KUKA KRL program: PROJET_PROFILO.src, PROJET_PROFILO.dat

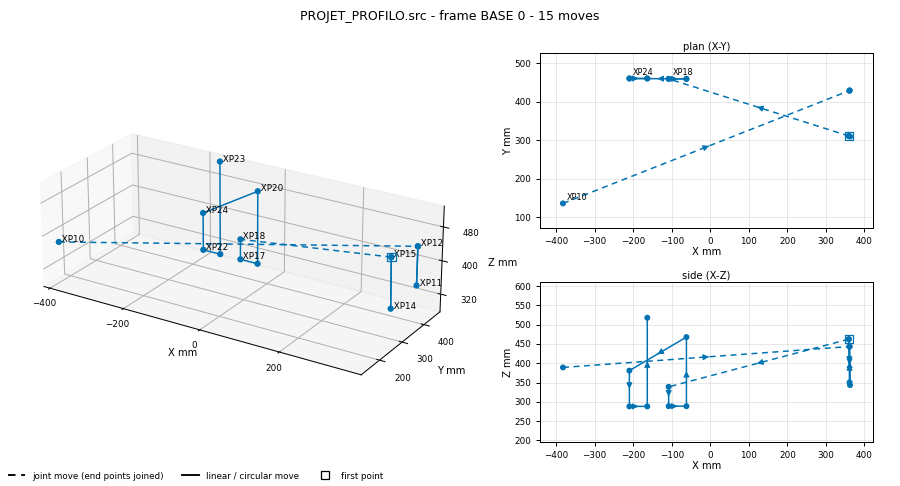
[picture p0: tool path of PROJET_PROFILO.src in frame BASE 0, 15 of 24 moves have a stored position in this frame; points joined in program order, loops and branches not executed]
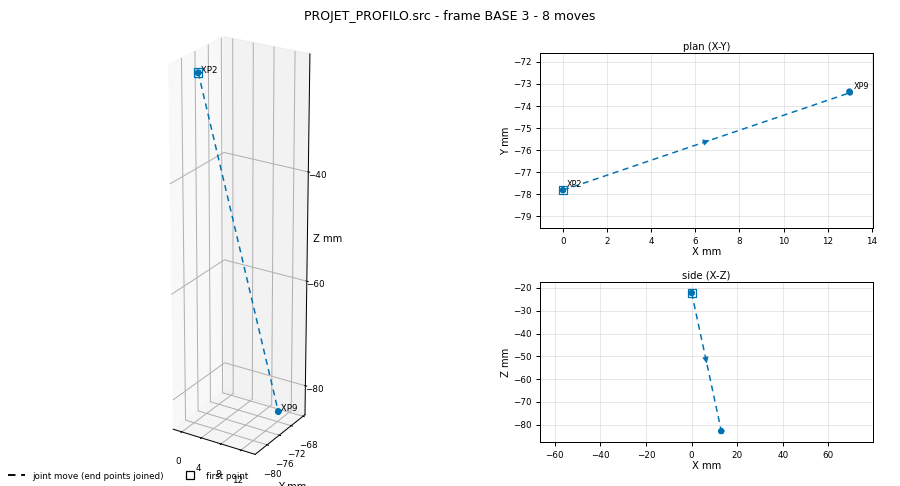
[picture p1: tool path of PROJET_PROFILO.src in frame BASE 3, 8 of 24 moves have a stored position in this frame; points joined in program order, loops and branches not executed]
--- PROJET_PROFILO.src ---
&ACCESS RVO
&REL 258
&PARAM TEMPLATE = C:\KRC\Roboter\Template\vorgabe
&PARAM EDITMASK = *
DEF PROJET_PROFILO( )
EXTFCT BOOL SEND(INT:OUT, STATE_T:OUT, STATE_T:OUT, MODUS_T:OUT)
EXTFCT BOOL RECEIVE(INT:OUT, STATE_T:OUT, STATE_T:OUT, MODUS_T:OUT, FRAME:OUT)
EXTFCT BOOL RECV_CHAR(INT:OUT, STATE_T:OUT, STATE_T:OUT, MODUS_T:OUT, CHAR:OUT)
EXTFCT BOOL RECV_DOUBLE(INT:OUT, STATE_T:OUT, STATE_T:OUT, MODUS_T:OUT, REAL:OUT)
EXTFCT BOOL SEND_CHAR(INT:OUT, STATE_T:OUT, STATE_T:OUT, MODUS_T:OUT, CHAR:IN)
EXTFCT BOOL PRENDRE_PROFILE(INT:OUT, STATE_T:OUT, STATE_T:OUT, MODUS_T:OUT, CHAR:OUT)

DECL INT HANDLE
DECL STATE_T SR_T
DECL STATE_T SC_T
DECL MODUS_T MR_T
DECL CHAR IN_CHAR
DECL CHAR OUT_CHAR
DECL BOOL R1

;FOLD INI
  ;FOLD BASISTECH INI
    GLOBAL INTERRUPT DECL 3 WHEN $STOPMESS==TRUE DO IR_STOPM ( )
    INTERRUPT ON 3
    BAS (#INITMOV,0 )
  ;ENDFOLD (BASISTECH INI)
  ;FOLD USER INI
    ;Make your modifications here

  ;ENDFOLD (USER INI)
;ENDFOLD (INI)
; initialization
IN_CHAR = " "
OUT_CHAR = " "
MR_T = #ABS

;FOLD PTP HOME  Vel= 10 % PDAT24;%{PE}%R 5.4.37,%MKUKATPBASIS,%CMOVE,%VPTP,%P 1:PTP, 2:HOME, 3:, 5:10, 7:PDAT24
$BWDSTART=FALSE
PDAT_ACT=PPDAT24
FDAT_ACT=FHOME
BAS(#PTP_PARAMS,10)
$H_POS=XHOME
PTP XHOME
;ENDFOLD

LOOP
;FOLD PULSE 27 'lacher'  State= TRUE   Time= 0.5 sec;%{PE}%R 5.4.37,%MKUKATPBASIS,%COUT,%VPULSE,%P 2:27, 3:lacher, 5:TRUE, 6:, 8:0.5
PULSE($OUT[27], TRUE,0.5)
;ENDFOLD
;FOLD WAIT Time= 1 sec;%{PE}%R 5.4.37,%MKUKATPBASIS,%CWAIT,%VWAIT,%P 2:1
WAIT SEC 1
;ENDFOLD
;FOLD PULSE 25 'prendre'  State= TRUE   Time= 0.5 sec;%{PE}%R 5.4.37,%MKUKATPBASIS,%COUT,%VPULSE,%P 2:25, 3:prendre, 5:TRUE, 6:, 8:0.5
PULSE($OUT[25], TRUE,0.5)
;ENDFOLD

; wait GO signal from PC
WHILE (IN_CHAR <> 71)
   R1 = RECV_CHAR(HANDLE, SR_T, SC_T, MR_T, IN_CHAR)
ENDWHILE

; go grab the cube
;FOLD PTP P15  Vel= 20 % PDAT28 Tool[3]:pince Base[0];%{PE}%R 5.4.37,%MKUKATPBASIS,%CMOVE,%VPTP,%P 1:PTP, 2:P15, 3:, 5:20, 7:PDAT28
$BWDSTART=FALSE
PDAT_ACT=PPDAT28
FDAT_ACT=FP15
BAS(#PTP_PARAMS,20)
PTP XP15
;ENDFOLD
;FOLD LIN P14  Vel= 0.1 m/s CPDAT18 Tool[3]:pince Base[0];%{PE}%R 5.4.37,%MKUKATPBASIS,%CMOVE,%VLIN,%P 1:LIN, 2:P14, 3:, 5:0.1, 7:CPDAT18
$BWDSTART=FALSE
LDAT_ACT=LCPDAT18
FDAT_ACT=FP14
BAS(#CP_PARAMS,0.1)
LIN XP14
;ENDFOLD
;FOLD PULSE 27 'lacher'  State= TRUE   Time= 0.5 sec;%{PE}%R 5.4.37,%MKUKATPBASIS,%COUT,%VPULSE,%P 2:27, 3:lacher, 5:TRUE, 6:, 8:0.5
PULSE($OUT[27], TRUE,0.5)
;ENDFOLD
;FOLD LIN P16  Vel= 0.2 m/s CPDAT19 Tool[3]:pince Base[0];%{PE}%R 5.4.37,%MKUKATPBASIS,%CMOVE,%VLIN,%P 1:LIN, 2:P16, 3:, 5:0.2, 7:CPDAT19
$BWDSTART=FALSE
LDAT_ACT=LCPDAT19
FDAT_ACT=FP16
BAS(#CP_PARAMS,0.2)
LIN XP16
;ENDFOLD

; cube taken, now go flip the cube
;FOLD PTP P18  Vel= 20 % PDAT29 Tool[3]:pince Base[0];%{PE}%R 5.4.37,%MKUKATPBASIS,%CMOVE,%VPTP,%P 1:PTP, 2:P18, 3:, 5:20, 7:PDAT29
$BWDSTART=FALSE
PDAT_ACT=PPDAT29
FDAT_ACT=FP18
BAS(#PTP_PARAMS,20)
PTP XP18
;ENDFOLD
;FOLD LIN P17  Vel= 0.1 m/s CPDAT20 Tool[3]:pince Base[0];%{PE}%R 5.4.37,%MKUKATPBASIS,%CMOVE,%VLIN,%P 1:LIN, 2:P17, 3:, 5:0.1, 7:CPDAT20
$BWDSTART=FALSE
LDAT_ACT=LCPDAT20
FDAT_ACT=FP17
BAS(#CP_PARAMS,0.1)
LIN XP17
;ENDFOLD
;FOLD PULSE 25 'prendre'  State= TRUE   Time= 0.5 sec;%{PE}%R 5.4.37,%MKUKATPBASIS,%COUT,%VPULSE,%P 2:25, 3:prendre, 5:TRUE, 6:, 8:0.5
PULSE($OUT[25], TRUE,0.5)
;ENDFOLD
;FOLD LIN P19  Vel= 0.1 m/s CPDAT21 Tool[3]:pince Base[0];%{PE}%R 5.4.37,%MKUKATPBASIS,%CMOVE,%VLIN,%P 1:LIN, 2:P19, 3:, 5:0.1, 7:CPDAT21
$BWDSTART=FALSE
LDAT_ACT=LCPDAT21
FDAT_ACT=FP19
BAS(#CP_PARAMS,0.1)
LIN XP19
;ENDFOLD
;FOLD LIN P20 CONT Vel= 0.1 m/s CPDAT24 Tool[3]:pince Base[0];%{PE}%R 5.4.37,%MKUKATPBASIS,%CMOVE,%VLIN,%P 1:LIN, 2:P20, 3:C_DIS, 5:0.1, 7:CPDAT24
$BWDSTART=FALSE
LDAT_ACT=LCPDAT24
FDAT_ACT=FP20
BAS(#CP_PARAMS,0.1)
LIN XP20 C_DIS
;ENDFOLD
;FOLD PULSE 27 'lacher'  State= TRUE   Time= 0.5 sec;%{PE}%R 5.4.37,%MKUKATPBASIS,%COUT,%VPULSE,%P 2:27, 3:lacher, 5:TRUE, 6:, 8:0.5
PULSE($OUT[27], TRUE,0.5)
;ENDFOLD
;FOLD LIN P24 CONT Vel= 0.1 m/s CPDAT26 Tool[3]:pince Base[0];%{PE}%R 5.4.37,%MKUKATPBASIS,%CMOVE,%VLIN,%P 1:LIN, 2:P24, 3:C_DIS, 5:0.1, 7:CPDAT26
$BWDSTART=FALSE
LDAT_ACT=LCPDAT26
FDAT_ACT=FP24
BAS(#CP_PARAMS,0.1)
LIN XP24 C_DIS
;ENDFOLD
;FOLD LIN P22  Vel= 0.1 m/s CPDAT25 Tool[3]:pince Base[0];%{PE}%R 5.4.37,%MKUKATPBASIS,%CMOVE,%VLIN,%P 1:LIN, 2:P22, 3:, 5:0.1, 7:CPDAT25
$BWDSTART=FALSE
LDAT_ACT=LCPDAT25
FDAT_ACT=FP22
BAS(#CP_PARAMS,0.1)
LIN XP22
;ENDFOLD
;FOLD LIN P21  Vel= 0.1 m/s CPDAT22 Tool[3]:pince Base[0];%{PE}%R 5.4.37,%MKUKATPBASIS,%CMOVE,%VLIN,%P 1:LIN, 2:P21, 3:, 5:0.1, 7:CPDAT22
$BWDSTART=FALSE
LDAT_ACT=LCPDAT22
FDAT_ACT=FP21
BAS(#CP_PARAMS,0.1)
LIN XP21
;ENDFOLD
;FOLD PULSE 25 'prendre'  State= TRUE   Time= 0.5 sec;%{PE}%R 5.4.37,%MKUKATPBASIS,%COUT,%VPULSE,%P 2:25, 3:prendre, 5:TRUE, 6:, 8:0.5
PULSE($OUT[25], TRUE,0.5)
;ENDFOLD
;FOLD LIN P23 CONT Vel= 0.1 m/s CPDAT23 Tool[3]:pince Base[0];%{PE}%R 5.4.37,%MKUKATPBASIS,%CMOVE,%VLIN,%P 1:LIN, 2:P23, 3:C_DIS, 5:0.1, 7:CPDAT23
$BWDSTART=FALSE
LDAT_ACT=LCPDAT23
FDAT_ACT=FP23
BAS(#CP_PARAMS,0.1)
LIN XP23 C_DIS
;ENDFOLD

; wait GO signal from PC
WHILE (IN_CHAR <> 71)
   R1 = RECV_CHAR(HANDLE, SR_T, SC_T, MR_T, IN_CHAR)
ENDWHILE

; go to points and take profiles
;FOLD PTP P2  Vel= 20 % PDAT19 Tool[3]:pince Base[3]:profilometre;%{PE}%R 5.4.37,%MKUKATPBASIS,%CMOVE,%VPTP,%P 1:PTP, 2:P2, 3:, 5:20, 7:PDAT19
$BWDSTART=FALSE
PDAT_ACT=PPDAT19
FDAT_ACT=FP2
BAS(#PTP_PARAMS,20)
PTP XP2
;ENDFOLD
R1 = PRENDRE_PROFILE(HANDLE, SR_T, SC_T, MR_T, IN_CHAR)
;FOLD PTP P6  Vel= 20 % PDAT20 Tool[3]:pince Base[3]:profilometre;%{PE}%R 5.4.37,%MKUKATPBASIS,%CMOVE,%VPTP,%P 1:PTP, 2:P6, 3:, 5:20, 7:PDAT20
$BWDSTART=FALSE
PDAT_ACT=PPDAT20
FDAT_ACT=FP6
BAS(#PTP_PARAMS,20)
PTP XP6
;ENDFOLD
R1 = PRENDRE_PROFILE(HANDLE, SR_T, SC_T, MR_T, IN_CHAR)
;FOLD PTP P7  Vel= 20 % PDAT21 Tool[3]:pince Base[3]:profilometre;%{PE}%R 5.4.37,%MKUKATPBASIS,%CMOVE,%VPTP,%P 1:PTP, 2:P7, 3:, 5:20, 7:PDAT21
$BWDSTART=FALSE
PDAT_ACT=PPDAT21
FDAT_ACT=FP7
BAS(#PTP_PARAMS,20)
PTP XP7
;ENDFOLD
R1 = PRENDRE_PROFILE(HANDLE, SR_T, SC_T, MR_T, IN_CHAR)
;FOLD PTP P8  Vel= 20 % PDAT22 Tool[3]:pince Base[3]:profilometre;%{PE}%R 5.4.37,%MKUKATPBASIS,%CMOVE,%VPTP,%P 1:PTP, 2:P8, 3:, 5:20, 7:PDAT22
$BWDSTART=FALSE
PDAT_ACT=PPDAT22
FDAT_ACT=FP8
BAS(#PTP_PARAMS,20)
PTP XP8
;ENDFOLD
R1 = PRENDRE_PROFILE(HANDLE, SR_T, SC_T, MR_T, IN_CHAR)

; upper face, scanned 4 times with different angles
;FOLD PTP P9  Vel= 20 % PDAT23 Tool[3]:pince Base[3]:profilometre;%{PE}%R 5.4.37,%MKUKATPBASIS,%CMOVE,%VPTP,%P 1:PTP, 2:P9, 3:, 5:20, 7:PDAT23
$BWDSTART=FALSE
PDAT_ACT=PPDAT23
FDAT_ACT=FP9
BAS(#PTP_PARAMS,20)
PTP XP9
;ENDFOLD
R1 = PRENDRE_PROFILE(HANDLE, SR_T, SC_T, MR_T, IN_CHAR)
;FOLD PTP P26  Vel= 20 % PDAT34 Tool[3]:pince Base[3]:profilometre;%{PE}%R 5.4.37,%MKUKATPBASIS,%CMOVE,%VPTP,%P 1:PTP, 2:P26, 3:, 5:20, 7:PDAT34
$BWDSTART=FALSE
PDAT_ACT=PPDAT34
FDAT_ACT=FP26
BAS(#PTP_PARAMS,20)
PTP XP26
;ENDFOLD
R1 = PRENDRE_PROFILE(HANDLE, SR_T, SC_T, MR_T, IN_CHAR)
;FOLD PTP P25  Vel= 20 % PDAT33 Tool[3]:pince Base[3]:profilometre;%{PE}%R 5.4.37,%MKUKATPBASIS,%CMOVE,%VPTP,%P 1:PTP, 2:P25, 3:, 5:20, 7:PDAT33
$BWDSTART=FALSE
PDAT_ACT=PPDAT33
FDAT_ACT=FP25
BAS(#PTP_PARAMS,20)
PTP XP25
;ENDFOLD
R1 = PRENDRE_PROFILE(HANDLE, SR_T, SC_T, MR_T, IN_CHAR)
;FOLD PTP P27  Vel= 20 % PDAT35 Tool[3]:pince Base[3]:profilometre;%{PE}%R 5.4.37,%MKUKATPBASIS,%CMOVE,%VPTP,%P 1:PTP, 2:P27, 3:, 5:20, 7:PDAT35
$BWDSTART=FALSE
PDAT_ACT=PPDAT35
FDAT_ACT=FP27
BAS(#PTP_PARAMS,20)
PTP XP27
;ENDFOLD
R1 = PRENDRE_PROFILE(HANDLE, SR_T, SC_T, MR_T, IN_CHAR)

; send EXIT to PC
R1 = SEND_CHAR(HANDLE, SR_T, SC_T, MR_T, 88)

; wait for PC tells part conform or not
WHILE (IN_CHAR <> 78) AND (IN_CHAR <> 89)
   R1 = RECV_CHAR(HANDLE, SR_T, SC_T, MR_T, IN_CHAR)
ENDWHILE

; part not conform
IF IN_CHAR == 78 THEN
;FOLD PTP P10  Vel= 20 % PDAT25 Tool[3]:pince Base[0];%{PE}%R 5.4.37,%MKUKATPBASIS,%CMOVE,%VPTP,%P 1:PTP, 2:P10, 3:, 5:20, 7:PDAT25
$BWDSTART=FALSE
PDAT_ACT=PPDAT25
FDAT_ACT=FP10
BAS(#PTP_PARAMS,20)
PTP XP10
;ENDFOLD
;FOLD PULSE 27 'lacher'  State= TRUE   Time= 0.5 sec;%{PE}%R 5.4.37,%MKUKATPBASIS,%COUT,%VPULSE,%P 2:27, 3:lacher, 5:TRUE, 6:, 8:0.5
PULSE($OUT[27], TRUE,0.5)
;ENDFOLD
ENDIF

; part conform
IF IN_CHAR == 89 THEN
;FOLD PTP P12  Vel= 20 % PDAT26 Tool[3]:pince Base[0];%{PE}%R 5.4.37,%MKUKATPBASIS,%CMOVE,%VPTP,%P 1:PTP, 2:P12, 3:, 5:20, 7:PDAT26
$BWDSTART=FALSE
PDAT_ACT=PPDAT26
FDAT_ACT=FP12
BAS(#PTP_PARAMS,20)
PTP XP12
;ENDFOLD
;FOLD LIN P11  Vel= 0.1 m/s CPDAT17 Tool[3]:pince Base[0];%{PE}%R 5.4.37,%MKUKATPBASIS,%CMOVE,%VLIN,%P 1:LIN, 2:P11, 3:, 5:0.1, 7:CPDAT17
$BWDSTART=FALSE
LDAT_ACT=LCPDAT17
FDAT_ACT=FP11
BAS(#CP_PARAMS,0.1)
LIN XP11
;ENDFOLD
;FOLD PULSE 27 'lacher'  State= TRUE   Time= 0.5 sec;%{PE}%R 5.4.37,%MKUKATPBASIS,%COUT,%VPULSE,%P 2:27, 3:lacher, 5:TRUE, 6:, 8:0.5
PULSE($OUT[27], TRUE,0.5)
;ENDFOLD
;FOLD LIN P13  Vel= 0.2 m/s CPDAT27 Tool[3]:pince Base[0];%{PE}%R 5.4.37,%MKUKATPBASIS,%CMOVE,%VLIN,%P 1:LIN, 2:P13, 3:, 5:0.2, 7:CPDAT27
$BWDSTART=FALSE
LDAT_ACT=LCPDAT27
FDAT_ACT=FP13
BAS(#CP_PARAMS,0.2)
LIN XP13
;ENDFOLD
ENDIF

ENDLOOP
END

--- PROJET_PROFILO.dat ---
&ACCESS RVO
&REL 258
&PARAM TEMPLATE = C:\KRC\Roboter\Template\vorgabe
&PARAM EDITMASK = *
DEFDAT  PROJET_PROFILO
;FOLD EXTERNAL DECLARATIONS;%{PE}%MKUKATPBASIS,%CEXT,%VCOMMON,%P
;FOLD BASISTECH EXT;%{PE}%MKUKATPBASIS,%CEXT,%VEXT,%P
EXT  BAS (BAS_COMMAND  :IN,REAL  :IN )
DECL INT SUCCESS
;ENDFOLD (BASISTECH EXT)
;FOLD USER EXT;%{E}%MKUKATPUSER,%CEXT,%VEXT,%P
;Make here your modifications

;ENDFOLD (USER EXT)
;ENDFOLD (EXTERNAL DECLERATIONS)
DECL BASIS_SUGG_T LAST_BASIS={POINT1[] "P27                     ",POINT2[] "P27                     ",CP_PARAMS[] "CPDAT26                 ",PTP_PARAMS[] "PDAT35                  ",CONT[] "                        ",CP_VEL[] "0.005                   ",PTP_VEL[] "20                      ",SPL_NAME[] "S0                      "}
DECL E6POS XP1={X 3.04208207,Y 411.683594,Z 361.17569,A 167.849899,B 89.528801,C 152.8974,S 2,T 43,E1 0.0,E2 0.0,E3 0.0,E4 0.0,E5 0.0,E6 0.0}
DECL FDAT FP1={TOOL_NO 2,BASE_NO 0,IPO_FRAME #BASE,POINT2[] " "}
DECL PDAT PPDAT1={VEL 100.0,ACC 100.0,APO_DIST 100.0}
DECL PDAT PPDAT2={VEL 100.0,ACC 100.0,APO_DIST 100.0}
DECL PDAT PPDAT3={VEL 100.0,ACC 100.0,APO_DIST 100.0}
DECL PDAT PPDAT4={VEL 100.0,ACC 100.0,APO_DIST 100.0}
DECL PDAT PPDAT5={VEL 100.0,ACC 100.0,APO_DIST 100.0}
DECL PDAT PPDAT6={VEL 100.0,ACC 100.0,APO_DIST 100.0}
DECL PDAT PPDAT7={VEL 100.0,ACC 100.0,APO_DIST 100.0}
DECL E6POS XP99={X -85.5281525,Y 414.985596,Z 387.865997,A 88.0866013,B 87.5991135,C 97.2242432,S 2,T 35,E1 0.0,E2 0.0,E3 0.0,E4 0.0,E5 0.0,E6 0.0}
DECL FDAT FP99={TOOL_NO 2,BASE_NO 0,IPO_FRAME #BASE,POINT2[] " "}
DECL PDAT PPDAT8={VEL 100.0,ACC 100.0,APO_DIST 100.0}
DECL INT LAST_XP_POINT=9
DECL E6POS XNEW_POINT={X -251.468094,Y 292.194702,Z 631.135681,A 91.6703262,B -87.1333008,C -129.946304,S 2,T 43,E1 0.0,E2 0.0,E3 0.0,E4 0.0,E5 0.0,E6 0.0}
DECL FDAT FNEW_POINT={TOOL_NO 0,BASE_NO 0,IPO_FRAME #BASE,POINT2[] " "}
DECL LDAT LCPDAT1={VEL 2.0,ACC 100.0,APO_DIST 100.0,APO_FAC 50.0,ORI_TYP #VAR}
DECL LDAT LCPDAT2={VEL 2.0,ACC 100.0,APO_DIST 100.0,APO_FAC 50.0,ORI_TYP #VAR}
DECL E6POS XINITIAL_POS={X 352.895111,Y 300.94281,Z 673.360901,A -90.7709427,B -1.56862795,C -179.936905,S 2,T 35,E1 0.0,E2 0.0,E3 0.0,E4 0.0,E5 0.0,E6 0.0}
DECL FDAT FINITIAL_POS={TOOL_NO 0,BASE_NO 0,IPO_FRAME #BASE,POINT2[] " "}
DECL PDAT PPDAT9={VEL 100.0,ACC 100.0,APO_DIST 100.0}
DECL PDAT PPDAT10={VEL 100.0,ACC 100.0,APO_DIST 100.0}
DECL LDAT LCPDAT3={VEL 2.0,ACC 100.0,APO_DIST 100.0,APO_FAC 50.0,ORI_TYP #VAR}
DECL LDAT LCPDAT4={VEL 2.0,ACC 100.0,APO_DIST 100.0,APO_FAC 50.0,ORI_TYP #VAR}
DECL LDAT LCPDAT5={VEL 2.0,ACC 100.0,APO_DIST 100.0,APO_FAC 50.0,ORI_TYP #VAR}
DECL LDAT LCPDAT6={VEL 2.0,ACC 100.0,APO_DIST 100.0,APO_FAC 50.0,ORI_TYP #VAR}
DECL LDAT LCPDAT7={VEL 2.0,ACC 100.0,APO_DIST 100.0,APO_FAC 50.0,ORI_TYP #VAR}
DECL E6POS XNEW_POINT_LIN_FAST={X -60.5829201,Y 419.159485,Z 498.605988,A 67.120079,B -2.27553606,C -179.295593,S 2,T 35,E1 0.0,E2 0.0,E3 0.0,E4 0.0,E5 0.0,E6 0.0}
DECL FDAT FNEW_POINT_LIN_FAST={TOOL_NO 0,BASE_NO 0,IPO_FRAME #BASE,POINT2[] " "}
DECL E6POS XNEW_POINT_LIN_SLOW={X -60.5829201,Y 419.159485,Z 498.605988,A 67.120079,B -2.27553606,C -179.295593,S 2,T 35,E1 0.0,E2 0.0,E3 0.0,E4 0.0,E5 0.0,E6 0.0}
DECL FDAT FNEW_POINT_LIN_SLOW={TOOL_NO 0,BASE_NO 0,IPO_FRAME #BASE,POINT2[] " "}
DECL PDAT PPDAT11={VEL 100.0,ACC 100.0,APO_DIST 100.0}
DECL PDAT PPDAT12={VEL 100.0,ACC 100.0,APO_DIST 100.0}
DECL LDAT LCPDAT8={VEL 2.0,ACC 100.0,APO_DIST 100.0,APO_FAC 50.0,ORI_TYP #VAR}
DECL LDAT LCPDAT9={VEL 2.0,ACC 100.0,APO_DIST 100.0,APO_FAC 50.0,ORI_TYP #VAR}
DECL PDAT PPDAT13={VEL 100.0,ACC 100.0,APO_DIST 100.0}
DECL E6POS XP2={X 0.00264483108,Y -77.8235779,Z -22.1945,A -153.933197,B -88.8520432,C 65.1572266,S 6,T 59,E1 0.0,E2 0.0,E3 0.0,E4 0.0,E5 0.0,E6 0.0}
DECL FDAT FP2={TOOL_NO 3,BASE_NO 3,IPO_FRAME #BASE,POINT2[] " "}
DECL PDAT PPDAT14={VEL 100.0,ACC 100.0,APO_DIST 100.0}
DECL E6POS XP3={X 0.211270601,Y 480.734589,Z 566.639587,A -94.440567,B 2.11090398,C 90.3766479,S 6,T 51,E1 0.0,E2 0.0,E3 0.0,E4 0.0,E5 0.0,E6 0.0}
DECL FDAT FP3={TOOL_NO 0,BASE_NO 0,IPO_FRAME #BASE,POINT2[] " "}
DECL LDAT LCPDAT10={VEL 2.0,ACC 100.0,APO_DIST 100.0,APO_FAC 50.0,ORI_TYP #VAR}
DECL E6POS XP4={X 0.211270601,Y 480.734589,Z 566.639587,A -94.440567,B 2.11090398,C 90.3766479,S 6,T 51,E1 0.0,E2 0.0,E3 0.0,E4 0.0,E5 0.0,E6 0.0}
DECL FDAT FP4={TOOL_NO 0,BASE_NO 0,IPO_FRAME #BASE,POINT2[] " "}
DECL LDAT LCPDAT11={VEL 2.0,ACC 100.0,APO_DIST 100.0,APO_FAC 50.0,ORI_TYP #VAR}
DECL E6POS XP5={X 47.832859,Y 50.5500603,Z -203.236404,A -94.440567,B 2.11090398,C 90.3766479,S 6,T 51,E1 0.0,E2 0.0,E3 0.0,E4 0.0,E5 0.0,E6 0.0}
DECL FDAT FP5={TOOL_NO 3,BASE_NO 3,IPO_FRAME #BASE,POINT2[] " "}
DECL LDAT LCPDAT12={VEL 2.0,ACC 100.0,APO_DIST 100.0,APO_FAC 50.0,ORI_TYP #VAR}
DECL E6POS XP6={X 0.00117324002,Y -77.8127594,Z -22.2087898,A -179.498199,B -0.486956209,C 91.2150726,S 6,T 27,E1 0.0,E2 0.0,E3 0.0,E4 0.0,E5 0.0,E6 0.0}
DECL FDAT FP6={TOOL_NO 3,BASE_NO 3,IPO_FRAME #BASE,POINT2[] " "}
DECL PDAT PPDAT15={VEL 100.0,ACC 100.0,APO_DIST 100.0}
DECL E6POS XP7={X 0.00117345597,Y -77.8127594,Z -22.2087898,A -19.7653904,B 88.5158768,C -108.539902,S 6,T 27,E1 0.0,E2 0.0,E3 0.0,E4 0.0,E5 0.0,E6 0.0}
DECL FDAT FP7={TOOL_NO 3,BASE_NO 3,IPO_FRAME #BASE,POINT2[] " "}
DECL PDAT PPDAT16={VEL 100.0,ACC 100.0,APO_DIST 100.0}
DECL E6POS XP8={X 0.00117460405,Y -77.8127594,Z -22.2087898,A -0.501615882,B 0.0515326709,C -88.7053375,S 6,T 59,E1 0.0,E2 0.0,E3 0.0,E4 0.0,E5 0.0,E6 0.0}
DECL FDAT FP8={TOOL_NO 3,BASE_NO 3,IPO_FRAME #BASE,POINT2[] " "}
DECL PDAT PPDAT17={VEL 100.0,ACC 100.0,APO_DIST 100.0}
DECL LDAT LCPDAT13={VEL 2.0,ACC 100.0,APO_DIST 100.0,APO_FAC 50.0,ORI_TYP #VAR}
DECL LDAT LCPDAT14={VEL 2.0,ACC 100.0,APO_DIST 100.0,APO_FAC 50.0,ORI_TYP #VAR}
DECL LDAT LCPDAT15={VEL 2.0,ACC 100.0,APO_DIST 100.0,APO_FAC 50.0,ORI_TYP #VAR}
DECL LDAT LCPDAT16={VEL 2.0,ACC 100.0,APO_DIST 100.0,APO_FAC 50.0,ORI_TYP #VAR}
DECL PDAT PPDAT18={VEL 100.0,ACC 100.0,APO_DIST 100.0}
DECL PDAT PPDAT19={VEL 100.0,ACC 100.0,APO_DIST 100.0}
DECL PDAT PPDAT20={VEL 100.0,ACC 100.0,APO_DIST 100.0}
DECL PDAT PPDAT21={VEL 100.0,ACC 100.0,APO_DIST 100.0}
DECL PDAT PPDAT22={VEL 100.0,ACC 100.0,APO_DIST 100.0}
DECL E6POS XP9={X 13.0152302,Y -73.394043,Z -82.7755432,A -175.600098,B 1.09652495,C 26.9111309,S 6,T 59,E1 0.0,E2 0.0,E3 0.0,E4 0.0,E5 0.0,E6 0.0}
DECL FDAT FP9={TOOL_NO 3,BASE_NO 3,IPO_FRAME #BASE,POINT2[] " "}
DECL PDAT PPDAT23={VEL 100.0,ACC 100.0,APO_DIST 100.0}
DECL PDAT PPDAT24={VEL 100.0,ACC 100.0,APO_DIST 100.0}
DECL E6POS XP10={X -382.229797,Y 136.348206,Z 389.157715,A 87.4006577,B -1.75323403,C -177.311707,S 6,T 59,E1 0.0,E2 0.0,E3 0.0,E4 0.0,E5 0.0,E6 0.0}
DECL FDAT FP10={TOOL_NO 3,BASE_NO 0,IPO_FRAME #BASE,POINT2[] " "}
DECL PDAT PPDAT25={VEL 100.0,ACC 100.0,APO_DIST 100.0}
DECL E6POS XP11={X 361.469086,Y 429.168213,Z 350.290985,A 89.2297974,B -0.773940682,C -179.077301,S 2,T 43,E1 0.0,E2 0.0,E3 0.0,E4 0.0,E5 0.0,E6 0.0}
DECL FDAT FP11={TOOL_NO 3,BASE_NO 0,IPO_FRAME #BASE,POINT2[] " "}
DECL LDAT LCPDAT17={VEL 2.0,ACC 100.0,APO_DIST 100.0,APO_FAC 50.0,ORI_TYP #VAR}
DECL E6POS XP12={X 361.442413,Y 429.135406,Z 443.394714,A 89.2239227,B -0.758097708,C -179.062393,S 2,T 43,E1 0.0,E2 0.0,E3 0.0,E4 0.0,E5 0.0,E6 0.0}
DECL FDAT FP12={TOOL_NO 3,BASE_NO 0,IPO_FRAME #BASE,POINT2[] " "}
DECL PDAT PPDAT26={VEL 100.0,ACC 100.0,APO_DIST 100.0}
DECL E6POS XP13={X 361.442413,Y 429.135406,Z 443.394714,A 89.2239227,B -0.758097708,C -179.062393,S 2,T 43,E1 0.0,E2 0.0,E3 0.0,E4 0.0,E5 0.0,E6 0.0}
DECL FDAT FP13={TOOL_NO 3,BASE_NO 0,IPO_FRAME #BASE,POINT2[] " "}
DECL PDAT PPDAT27={VEL 100.0,ACC 100.0,APO_DIST 100.0}
DECL E6POS XP14={X 362.679688,Y 309.753906,Z 343.361603,A 179.220901,B -0.79322809,C 179.790802,S 2,T 43,E1 0.0,E2 0.0,E3 0.0,E4 0.0,E5 0.0,E6 0.0}
DECL FDAT FP14={TOOL_NO 3,BASE_NO 0,IPO_FRAME #BASE,POINT2[] " "}
DECL LDAT LCPDAT18={VEL 2.0,ACC 100.0,APO_DIST 100.0,APO_FAC 50.0,ORI_TYP #VAR}
DECL E6POS XP15={X 359.65799,Y 311.270905,Z 462.464996,A 179.216599,B -0.798424482,C 179.8069,S 2,T 43,E1 0.0,E2 0.0,E3 0.0,E4 0.0,E5 0.0,E6 0.0}
DECL FDAT FP15={TOOL_NO 3,BASE_NO 0,IPO_FRAME #BASE,POINT2[] " "}
DECL PDAT PPDAT28={VEL 100.0,ACC 100.0,APO_DIST 100.0}
DECL E6POS XP16={X 359.65799,Y 311.270905,Z 462.464996,A 179.216599,B -0.798424482,C 179.8069,S 2,T 43,E1 0.0,E2 0.0,E3 0.0,E4 0.0,E5 0.0,E6 0.0}
DECL FDAT FP16={TOOL_NO 3,BASE_NO 0,IPO_FRAME #BASE,POINT2[] " "}
DECL LDAT LCPDAT19={VEL 2.0,ACC 100.0,APO_DIST 100.0,APO_FAC 50.0,ORI_TYP #VAR}
DECL E6POS XP17={X -107.957001,Y 459.539398,Z 288.618195,A -89.8100433,B -0.0262975805,C 91.8582687,S 2,T 11,E1 0.0,E2 0.0,E3 0.0,E4 0.0,E5 0.0,E6 0.0}
DECL FDAT FP17={TOOL_NO 3,BASE_NO 0,IPO_FRAME #BASE,POINT2[] " "}
DECL LDAT LCPDAT20={VEL 2.0,ACC 100.0,APO_DIST 100.0,APO_FAC 50.0,ORI_TYP #VAR}
DECL E6POS XP18={X -107.951401,Y 459.55069,Z 338.765594,A -89.8116684,B -0.0291104,C 91.8583374,S 2,T 11,E1 0.0,E2 0.0,E3 0.0,E4 0.0,E5 0.0,E6 0.0}
DECL FDAT FP18={TOOL_NO 3,BASE_NO 0,IPO_FRAME #BASE,POINT2[] " "}
DECL PDAT PPDAT29={VEL 100.0,ACC 100.0,APO_DIST 100.0}
DECL E6POS XP19={X -61.8498192,Y 459.524506,Z 288.55069,A -89.8078079,B -0.0331712812,C 91.8604126,S 2,T 11,E1 0.0,E2 0.0,E3 0.0,E4 0.0,E5 0.0,E6 0.0}
DECL FDAT FP19={TOOL_NO 3,BASE_NO 0,IPO_FRAME #BASE,POINT2[] " "}
DECL LDAT LCPDAT21={VEL 2.0,ACC 100.0,APO_DIST 100.0,APO_FAC 50.0,ORI_TYP #VAR}
DECL E6POS XP20={X -61.852829,Y 459.462006,Z 467.888,A -89.7964706,B -0.0613530986,C 91.8438721,S 2,T 11,E1 0.0,E2 0.0,E3 0.0,E4 0.0,E5 0.0,E6 0.0}
DECL FDAT FP20={TOOL_NO 3,BASE_NO 0,IPO_FRAME #BASE,POINT2[] " "}
DECL PDAT PPDAT30={VEL 100.0,ACC 100.0,APO_DIST 100.0}
DECL E6POS XP21={X -163.422806,Y 460.499115,Z 288.062714,A -90.2210999,B -0.260996312,C -90.0108871,S 2,T 35,E1 0.0,E2 0.0,E3 0.0,E4 0.0,E5 0.0,E6 0.0}
DECL FDAT FP21={TOOL_NO 3,BASE_NO 0,IPO_FRAME #BASE,POINT2[] " "}
DECL PDAT PPDAT31={VEL 100.0,ACC 100.0,APO_DIST 100.0}
DECL LDAT LCPDAT22={VEL 2.0,ACC 100.0,APO_DIST 100.0,APO_FAC 50.0,ORI_TYP #VAR}
DECL E6POS XP22={X -209.9021,Y 460.505402,Z 288.060791,A -90.2218399,B -0.259503812,C -90.014267,S 2,T 35,E1 0.0,E2 0.0,E3 0.0,E4 0.0,E5 0.0,E6 0.0}
DECL FDAT FP22={TOOL_NO 3,BASE_NO 0,IPO_FRAME #BASE,POINT2[] " "}
DECL PDAT PPDAT32={VEL 100.0,ACC 100.0,APO_DIST 100.0}
DECL E6POS XP23={X -163.408005,Y 460.491699,Z 518.076904,A -74.2553406,B -0.993976772,C -90.0108871,S 6,T 59,E1 0.0,E2 0.0,E3 0.0,E4 0.0,E5 0.0,E6 0.0}
DECL FDAT FP23={TOOL_NO 3,BASE_NO 0,IPO_FRAME #BASE,POINT2[] " "}
DECL LDAT LCPDAT23={VEL 2.0,ACC 100.0,APO_DIST 100.0,APO_FAC 50.0,ORI_TYP #VAR}
DECL LDAT LCPDAT24={VEL 2.0,ACC 100.0,APO_DIST 100.0,APO_FAC 50.0,ORI_TYP #VAR}
DECL LDAT LCPDAT25={VEL 2.0,ACC 100.0,APO_DIST 100.0,APO_FAC 50.0,ORI_TYP #VAR}
DECL E6POS XP24={X -209.904907,Y 460.509094,Z 380.869293,A -82.867569,B -0.251814306,C -90.0270767,S 2,T 35,E1 0.0,E2 0.0,E3 0.0,E4 0.0,E5 0.0,E6 0.0}
DECL FDAT FP24={TOOL_NO 3,BASE_NO 0,IPO_FRAME #BASE,POINT2[] " "}
DECL LDAT LCPDAT26={VEL 2.0,ACC 100.0,APO_DIST 100.0,APO_FAC 50.0,ORI_TYP #VAR}
DECL LDAT LCPDAT27={VEL 2.0,ACC 100.0,APO_DIST 100.0,APO_FAC 50.0,ORI_TYP #VAR}
DECL E6POS XP25={X 12.9849701,Y -73.3447723,Z -82.8352127,A 5.58934498,B -0.501115322,C -26.9344196,S 6,T 27,E1 0.0,E2 0.0,E3 0.0,E4 0.0,E5 0.0,E6 0.0}
DECL FDAT FP25={TOOL_NO 3,BASE_NO 3,IPO_FRAME #BASE,POINT2[] " "}
DECL PDAT PPDAT33={VEL 100.0,ACC 100.0,APO_DIST 100.0}
DECL E6POS XP26={X 12.9980803,Y -73.3662796,Z -82.8090973,A 93.7982483,B 26.9083691,C -1.25471699,S 6,T 27,E1 0.0,E2 0.0,E3 0.0,E4 0.0,E5 0.0,E6 0.0}
DECL FDAT FP26={TOOL_NO 3,BASE_NO 3,IPO_FRAME #BASE,POINT2[] " "}
DECL PDAT PPDAT34={VEL 100.0,ACC 100.0,APO_DIST 100.0}
DECL E6POS XP27={X 12.9902201,Y -73.3393021,Z -82.8367767,A -84.5559998,B -26.9351501,C 0.512929678,S 6,T 27,E1 0.0,E2 0.0,E3 0.0,E4 0.0,E5 0.0,E6 0.0}
DECL FDAT FP27={TOOL_NO 3,BASE_NO 3,IPO_FRAME #BASE,POINT2[] " "}
DECL PDAT PPDAT35={VEL 100.0,ACC 100.0,APO_DIST 100.0}
ENDDAT
